FUNCTION_BLOCK DriveControl
VAR
    isHardwareEnabled : BOOL;
    targetVelocity  : REAL;
END_VAR
VAR_OUTPUT
END_VAR
VAR
END_VAR

METHOD Enable : BOOL
VAR_INPUT
END_VAR
isHardwareEnabled := TRUE;
END_METHOD

METHOD MoveVelocity : BOOL
VAR_INPUT
    inVelocity : REAL;
END_VAR
targetVelocity:= inVelocity;
END_METHOD

METHOD QuickStop : BOOL
VAR_INPUT
END_VAR
targetVelocity := 0;
isHardwareEnabled := FALSE;
END_METHOD

END_FUNCTION_BLOCK

(* stored: Version 1.1.0.1, ProductVersion 3.1.4024.16
   POU DriveControl: Id {8e21d231-1779-4792-ad64-990034fa470d}, SpecialFunc None
   Method Enable: Id {3e2778b0-851d-4739-8690-9c412d5b2175}
   Method MoveVelocity: Id {56164e5b-7099-494c-8b8c-899f46d97fe6}
   Method QuickStop: Id {0f40a846-a15f-4b05-a355-8a65eb0f8462} *)
